{attribute addProperty BoxType "EL7041-0001-0017"}
{attribute addProperty Id "ENC_Status_compactAT %I*ENC_Status_compact_58C6E2B94860STM_StatusAT %I*STM_Status_817C32CB1620ENC_Control_compactAT %Q*ENC_Control_compact_03701F333240STM_ControlAT %Q*STM_Control_91ECC2DE1620STM_VelocityAT %Q*STM_Velocity_1D89B5C21620WcStateAT %I*WcState_F855686C1620InfoDataAT %I*InfoData_6C7DEEF988110"}
{attribute addProperty CRC "1102109544"}
{attribute addProperty SizeInBites "232"}
{attribute addProperty SizeInBytes "29"}
TYPE EL7041_41EBDE37 :
STRUCT
	{attribute addProperty Name "ENC_Status_compact"}
	ENC_Status_compact : ENC_Status_compact_58C6E2B9;
	{attribute addProperty Name "STM_Status"}
	STM_Status : STM_Status_817C32CB;
	{attribute addProperty Name "ENC_Control_compact"}
	ENC_Control_compact : ENC_Control_compact_03701F33;
	{attribute addProperty Name "STM_Control"}
	STM_Control : STM_Control_91ECC2DE;
	{attribute addProperty Name "STM_Velocity"}
	STM_Velocity : STM_Velocity_1D89B5C2;
	{attribute addProperty Name "WcState"}
	WcState : WcState_F855686C;
	{attribute addProperty Name "InfoData"}
	InfoData : InfoData_6C7DEEF9;
END_STRUCT
END_TYPE

(* stored: Version 1.2.0.0, ProductVersion 3.1.4024.9
   DUT EL7041_41EBDE37: Id {40d1d72f-9c1b-4473-a773-6ef0140eec56} *)
